{attribute 'linkalways'} 
{attribute 'no_explicit_call' := 'This FB is a CLASS and must be accessed using methods or properties'}
{attribute 'enable_dynamic_creation'}
FUNCTION_BLOCK FINAL LT_REAL EXTENDS Node
VAR
	in1 : _REAL(0.0);
	in2 : _REAL(0.0);
	out : _BOOL(FALSE);
END_VAR

METHOD PUBLIC Clone : I_Node
VAR
	pNode : POINTER TO LT_REAL;
END_VAR
pNode := __NEW(LT_REAL);
Clone := pNode^;
END_METHOD

METHOD FB_init : BOOL
VAR_INPUT
	bInitRetains : BOOL; // if TRUE, the retain variables are initialized (warm start / cold start)
	bInCopyCode : BOOL;  // if TRUE, the instance afterwards gets moved into the copy code (online change)
END_VAR
AddInput('in1',THIS^.in1);
AddInput('in2',THIS^.in2);
AddOutput('out', THIS^.out);
END_METHOD

METHOD PROTECTED OnExecute
VAR
END_VAR
out.Value := in1.Value < in2.Value;
END_METHOD

END_FUNCTION_BLOCK

(* stored: Version 1.1.0.1, ProductVersion 3.1.4024.15
   POU LT_REAL: Id {78ae08a9-618c-41c4-a5ec-57d905f070bc}, SpecialFunc None
   Folder Constructor: Id {be397ce9-1ddd-4897-a885-a6d48cf5e9d0}
   Method Clone: Id {2918c533-bbae-425b-9524-c3d5722178fe}
   Method FB_init: Id {e1e59d5f-63ad-48a8-bcee-21ce209bccf0}
   Method OnExecute: Id {d5b79815-6683-40de-8196-478c6d0e4898} *)
